FUNCTION_BLOCK Fb_SafetyCheck
VAR_INPUT
END_VAR
VAR_OUTPUT
END_VAR
VAR
	i, j:INT;
	m_checkDelay :ARRAY[1..g_maxNum] OF checkDelay;
	m_checkDelayTime :checkDelayTime;
	m_checkPermit:ARRAY[1..g_maxNum] OF  checkPermit;
	
	m_jntErrFlag:ARRAY[1..g_maxNum,0..g_maxArmJoint,1..3] OF BOOL;
	m_armErrFlag:ARRAY [1..g_maxNum,1..3] OF BOOL;
	m_errCode:UDINT;
	m_resetFlag : BOOL:= FALSE;
	m_resetFlagTon : TON;
	
	m_errNumType: ARRAY [1..3] OF INT;
	m_ArrayErrCodeType:ARRAY [1..3] OF ARRAY [0..100] OF UDINT;
	
	//The fault is sent to the UI at the frequency of 0.1S
	m_errCodeUpdateFlag: ARRAY [1..3] OF BOOL;
	m_errCodeUpdateTon: ARRAY [1..3] OF TON;
	
	m_curJntTorqueIOlast :ARRAY [1..g_maxArmNum] OF vec7di;  
	m_cmdJntPosLast : ARRAY [1..g_maxArmNum] OF vec7d;  
	m_cartCurJntTorqueIOlast :ARRAY [1..4] OF LREAL;  
	m_cartCmdJntPosLast : ARRAY [1..4] OF LREAL; 
	o_ErrCode:ARRAY [1..3] OF UDINT;
		
	//error robot data record
	m_dataRecord : Fb_dataRecord;
	
	m_PromptMassBusy:BOOL;
	m_PromptFlag:ARRAY[1..g_maxNum,1..20] OF UINT;
	m_deleteCode:UDINT;
	m_EtherCATCheck :ARRAY [1..g_mArmNum] OF Fb_EtherCATCheck;
	
	//drive  heartbeat single check
	m_heartbeatCheck :ARRAY [1..g_maxNum] OF ARRAY [1..g_maxArmJoint] OF FB_HeartbeatDetect;
	m_bHeartbeatCheck : ARRAY [1..g_maxNum] OF ARRAY [1..g_maxArmJoint] OF BOOL;
END_VAR


VAR CONSTANT
	m_codeUpdateDelay:TIME:=T#0.1S;
	
	//Fault level: 1 indicates  prompt message, 2 indicates a recoverable fault and 3 indicates an unrecoverable fault
	m_promptMessageLevel : UINT :=1;
	m_rcvLevel : UINT :=2;
	m_unrcvLevel : UINT :=3;
END_VAR


METHOD armSafetyCheck : BOOL
VAR_INPUT
	i_armId:INT;
	i_safetyCheckVar :ARRAY[1..g_maxNum] OF checkInputVariable;
	i_masterStatus :ST_MasterStatus;
	i_masterJointData : ST_MasterJointData;
END_VAR

VAR
	k:INT;
	motorHallCheck : UDINT;
	motorPhaseCheck : UDINT;
	motorDriveError : BOOL;
	lossCommuniJoint : INT;
END_VAR
//驱动器状态监测、驱动器未连接
FOR i:=1 TO g_mJntNum BY 1 DO
	m_bHeartbeatCheck[i_armId][i] := TRUE;//m_heartbeatCheck[i_armId][i].run(i_safetyCheckVar[i_armId].m_masterDriverInput[i].m_heartBeat);
	m_checkDelay[i_armId].T_jntStatusErr[i](IN:= (i_safetyCheckVar[i_armId].m_masterDriverInput[i].m_statusWord=0 AND m_checkPermit[i_armId].m_jntStatusErr[i]), PT:=m_checkDelayTime.Ti_jntStatusErr , Q=> , ET=> );
	IF m_checkDelay[i_armId].T_jntStatusErr[i].Q OR NOT m_bHeartbeatCheck[i_armId][i] THEN
		errCodeAssign(i_armId, i_armId,  0, i, 16#3002 ,m_unrcvLevel );
		EXIT;
	END_IF
END_FOR



//关节编码器监测
FOR i:=1 TO g_mJntNum BY 1 DO	
	IF i = 2 THEN
		//m_checkDelay[i_ArmId].T_linkEncErrCode[i](IN:= (driveErrorCheck(i_armId, i, 1, i_safetyCheckVar[i_ArmId].m_masterDriverInput[4].m_driverError) > 0  AND m_checkPermit[i_ArmId].m_linkEncErr[i]), PT:=m_checkDelayTime.Ti_linkEncErrCode , Q=> , ET=> );
	ELSE
		//m_checkDelay[i_ArmId].T_linkEncErrCode[i](IN:= (driveErrorCheck(i_armId, i, 1, i_safetyCheckVar[i_ArmId].m_masterDriverInput[i].m_driverError) > 0  AND m_checkPermit[i_ArmId].m_linkEncErr[i]), PT:=m_checkDelayTime.Ti_linkEncErrCode , Q=> , ET=> );
	END_IF
	m_checkDelay[i_ArmId].T_linkEncErr[i](IN:= (i_safetyCheckVar[i_ArmId].m_masterDriverInput[i].m_linkEncoder=g_maxLinkEnc OR i_safetyCheckVar[i_ArmId].m_masterDriverInput[i].m_linkEncoder=g_minLinkEnc) AND m_checkPermit[i_ArmId].m_linkEncErr[i], PT:=m_checkDelayTime.Ti_linkEncErr , Q=> , ET=> );
	IF m_checkDelay[i_ArmId].T_linkEncErr[i].Q OR m_checkDelay[i_ArmId].T_linkEncErrCode[i].Q THEN
		errCodeAssign(i_ArmId, i_ArmId,  0, i,  16#3003 ,m_unrcvLevel );
	END_IF
END_FOR


//驱动器错误检测
//FOR i:=1 TO g_mJntNum BY 1 DO
//	m_checkDelay[i_ArmId].T_DriveErr[i](IN:= (i_safetyCheckVar[i_ArmId].m_masterDriverInput[i].m_driverError AND g_driveErrWord)=g_driveErrWord AND m_checkPermit[i_ArmId].m_driveErr[i] , PT:=m_checkDelayTime.Ti_driveErr , Q=> , ET=> );
//	IF m_checkDelay[i_ArmId].T_DriveErr[i].Q THEN
//		errCodeAssign(i_ArmId, i_ArmId,  0, i, 16#3004 ,m_unrcvLevel );
//	END_IF
//END_FOR


//双编码器偏差过大检测
FOR i:=1 TO g_mJntNum BY 1 DO
	m_checkDelay[i_ArmId].T_armJntEncErr[i](IN:= ABS(i_masterJointData.m_curLinkPos[i_armId][i]-i_masterJointData.m_curJntPos[i_armId][i])>=g_armMaxJntEncErr[i] AND m_checkPermit[i_ArmId].m_armJntEncErr[i], PT:=m_checkDelayTime.Ti_armJntEncErr , Q=> , ET=> );
	IF m_checkDelay[i_ArmId].T_armJntEncErr[i].Q THEN
		errCodeAssign( i_ArmId, i_ArmId,  0, i, 16#3005, m_unrcvLevel );
	END_IF
END_FOR


//关节运动超限位
FOR i:=1 TO g_mJntNum BY 1 DO
	m_checkDelay[i_armId].T_outOfLimit[i](IN:= (i_masterJointData.m_curJntPos[i_armId][i]>= (g_maxJntPos[i_armId,i] + g_armJntPosLimitBuffer[i]) OR i_masterJointData.m_curJntPos[i_armId][i]<=(g_minJntPos[i_armId,i] - g_armJntPosLimitBuffer[i])) AND m_checkPermit[i_ArmId].m_outOfLimit[i], PT:=m_checkDelayTime.Ti_outofLimit , Q=> , ET=> );
	IF m_checkDelay[i_armId].T_outOfLimit[i].Q THEN
		errCodeAssign(i_armId, i_ArmId,  0, i, 16#3006, m_unrcvLevel );
	END_IF
END_FOR

//check motor hall single, error code 27
FOR i:=1 TO g_mJntNum DO
	motorHallCheck := driveErrorCheck(i_armId, i, 2, i_safetyCheckVar[i_ArmId].m_masterDriverInput[i].m_driverError);		
	m_checkDelay[i_ArmId].T_motorHallCheck[i](IN:= (motorHallCheck  = 1) , PT:=m_checkDelayTime.Ti_motorHallCheck , Q=> , ET=> );
	IF  m_checkDelay[i_ArmId].T_motorHallCheck[i].Q THEN
		errCodeAssign(i_ArmId, i_ArmId,  0, i, 16#300B ,m_unrcvLevel );
	END_IF
END_FOR


//check motor phase single, error code 30
FOR i:=1 TO g_mJntNum DO
	motorPhaseCheck := driveErrorCheck(i_armId, i, 3, i_safetyCheckVar[i_ArmId].m_masterDriverInput[i].m_driverError);		
	m_checkDelay[i_ArmId].T_motorPhaseCheck[i](IN:= (motorPhaseCheck  = 1) , PT:=m_checkDelayTime.Ti_motorPhaseCheck , Q=> , ET=> );
	IF  m_checkDelay[i_ArmId].T_motorPhaseCheck[i].Q THEN
		errCodeAssign(i_ArmId, i_ArmId,  0, i, 16#300C ,m_unrcvLevel );
	END_IF
END_FOR


//check motor drive, error code 31
FOR i:=1 TO g_mJntNum DO
	motorDriveError := (i_safetyCheckVar[i_ArmId].m_masterDriverInput[i].m_driverError AND 16#80000000)=16#80000000;
	m_checkDelay[i_ArmId].T_motorDriveError[i](IN:= motorDriveError, PT:=m_checkDelayTime.Ti_motorDriveCheck , Q=> , ET=> );
	IF  m_checkDelay[i_ArmId].T_motorDriveError[i].Q THEN
		errCodeAssign(i_ArmId, i_ArmId,  0, i, 16#300D ,m_unrcvLevel );
	END_IF
END_FOR


//关节跟随误差过大
FOR i:=1 TO g_mJntNum BY 1 DO
	m_checkDelay[i_ArmId].T_armJntFollowErr[i](IN:= ABS(i_masterJointData.m_cmdJntPos[i_armId][i]- i_masterJointData.m_curJntPos[i_armId][i])>g_armMaxJntFollowErr[i]  AND m_checkPermit[i_ArmId].m_armJntFollowErr[i], PT:=m_checkDelayTime.Ti_armJntFollowErr , Q=> , ET=> );
	IF m_checkDelay[i_ArmId].T_armJntFollowErr[i].Q THEN
		errCodeAssign(i_ArmId, i_ArmId,  0, i, 16#2002, m_rcvLevel );
	END_IF
END_FOR


//笛卡尔空间指令与位置偏差检测
//FOR i:=1 TO 6 BY 1 DO
//	m_checkDelay[i_ArmId].T_spacePoseErr[i](IN:= i_safetyCheckVar[i_ArmId].m_spacePoseErr[i]> g_maxCartPoseErr[i] AND m_checkPermit[i_ArmId].m_spacePoseErr[i], PT:=m_checkDelayTime.Ti_spacePoseErr , Q=> , ET=> );
//	IF m_checkDelay[i_ArmId].T_spacePoseErr[i].Q THEN
//		errCodeAssign(i_ArmId, i_ArmId, 1, i, 16#2004, m_rcvLevel );
//	END_IF
//END_FOR


//current overrun check
FOR i:=1 TO g_mJntNum BY 1 DO
	m_checkDelay[i_armId].T_jntCurrentErr[i](IN:= ABS(i_safetyCheckVar[i_armId].m_motorCurrentIntegral[i])>g_motorCurrentLimit[i] AND m_checkPermit[i_ArmId].m_jntCurrentErr[i], PT:=m_checkDelayTime.Ti_jntCurrentErr , Q=> , ET=> );
	IF m_checkDelay[i_armId].T_jntCurrentErr[i].Q THEN
		errCodeAssign(i_armId, i_ArmId,  0, i, 16#2005, m_rcvLevel );
	END_IF
END_FOR


//Ethercat communication check
lossCommuniJoint := g_maxArmJoint;
FOR i:=1 TO g_mJntNum BY 1 DO
	IF NOT i_safetyCheckVar[i_ArmId].m_EtherCATState[i].EtherCATState THEN
		lossCommuniJoint := MIN(lossCommuniJoint,i);
		errCodeAssign(i_ArmId, i_ArmId, 0, lossCommuniJoint, 16#2006, m_rcvLevel );
		IF i > lossCommuniJoint THEN
			m_jntErrFlag[i_armId,i,m_rcvLevel]:=TRUE;
		END_IF
	END_IF
END_FOR


//self check failure
IF i_masterStatus.m_armState[i_armId] = MasterArmState_Home AND i_masterStatus.m_timePeriod[i] > g_selfCheckTimeLimit THEN//i_safetyCheckVar[i_armId].m_selfCheckFail THEN
	errCodeAssign(i_armId, i_ArmId,  0, 0, 16#2010, m_rcvLevel );
END_IF

//motor encoder mutation detection
FOR i:=1 TO g_mJntNum BY 1 DO
	IF i_safetyCheckVar[i_armId].m_motorEncSaltaValue[i]>g_maxJntCurSalta[i] THEN
		errCodeAssign(i_armId, i_ArmId, 0, i, 16#200C, m_rcvLevel );
	END_IF
END_FOR

//master hall anomaly
IF i_masterStatus.m_gripHallSensor[i_armId] = 0 THEN
	errCodeAssign(i_armId, i_ArmId, 0, 0, 16#200E, m_rcvLevel );
END_IF

//drive Ethercat CRC lost
FOR i:=1 TO g_mJntNum BY 1 DO
	IF (i_safetyCheckVar[i_armId].m_EtherCATState[i].CRCPortA)>m_minLossFrame OR  (i_safetyCheckVar[i_armId].m_EtherCATState[i].CRCPortB)>m_minLossFrame OR  (i_safetyCheckVar[i_armId].m_EtherCATState[i].CRCPortC)>m_minLossFrame  THEN
		errCodeAssign(i_armId, i_ArmId, 0, i, 16#200F, m_rcvLevel );
	END_IF
END_FOR
END_METHOD

METHOD arrayDeleteFrist : ARRAY [0..100] OF UDINT;
VAR_INPUT
	i_array:ARRAY [0..100] OF UDINT;
END_VAR

VAR
	k:INT;
END_VAR

arrayDeleteFrist[100]:=0;

FOR k:=0 TO 99 BY 1 DO
	arrayDeleteFrist[k]:=i_array[k+1];
END_FOR
END_METHOD

METHOD arrayDeleteInput : BOOL
VAR_INPUT
	i_Array:ARRAY[0..100] OF UDINT;
	i_DeleteCode:UDINT;
END_VAR

VAR_OUTPUT
	o_Array:ARRAY[0..100] OF UDINT;
	
END_VAR

VAR
	i:INT;
	Falg:BOOL;
END_VAR

FOR i:=0 TO 20 BY 1 DO 
	IF i_Array[i]=i_DeleteCode THEN
		Falg:=TRUE;
	END_IF
	
	IF Falg=TRUE THEN
		o_Array[i]:=i_Array[i+1];
	ELSE
		o_Array[i]:=i_Array[i];
	END_IF
END_FOR
o_Array[20]:=0;
END_METHOD

METHOD arrayFIFO : ARRAY [0..100] OF  UDINT
VAR_INPUT
	i_array:ARRAY[0..100] OF UDINT;
	i_newData:UDINT;
END_VAR

VAR
	i:INT;
END_VAR

FOR i:=0 TO 20 BY 1 DO
	arrayFIFO[i+1]:=i_array[i];
END_FOR

arrayFIFO[0]:=i_newData;
END_METHOD

METHOD arrayFILO : ARRAY [0..100] OF  UDINT
VAR_INPUT
	i_array:ARRAY[0..100] OF UDINT;
	i_newData:UDINT;
END_VAR

VAR
	i:INT;
END_VAR

FOR i:=0 TO 99 BY 1 DO
	arrayFILO[i]:=i_array[i];
	IF i_array[i]=0 THEN
		arrayFILO[i]:=i_newData;
		EXIT;
	END_IF
END_FOR
END_METHOD

METHOD cartSafetyCheck : BOOL
VAR_INPUT
	i_armId:INT;
	i_safetyCheckVar : checkInputVariable;
	i_cartJointData : ST_CartJointData;
END_VAR


VAR
	k:INT;
	motorHallCheck : UDINT;
	motorPhaseCheck : UDINT;
	motorDriveError : BOOL;
	lossCommuniJoint : INT;
END_VAR
//驱动器状态监测、驱动器未连接
FOR i:=1 TO g_maxCartJoint BY 1 DO
	m_bHeartbeatCheck[i_armId][i] := TRUE;//m_heartbeatCheck[i_armId][i].run(i_safetyCheckVar.m_cartDriverInput[i].m_heartBeat);
	m_checkDelay[i_armId].T_cartJntStatusErr[i](IN:= (i_safetyCheckVar.m_cartDriverInput[i].m_statusWord=0 AND m_checkPermit[i_ArmId].m_cartJntStatus[i]), PT:=m_checkDelayTime.Ti_CarJntStatus , Q=> , ET=> );
	IF m_checkDelay[i_armId].T_cartJntStatusErr[i].Q OR NOT m_bHeartbeatCheck[i_armId][i] THEN
		errCodeAssign(i_armId, i_ArmId,  0, i, 16#3002 ,m_unrcvLevel );
	END_IF
END_FOR



//关节编码器监测
FOR i:=1 TO g_maxCartJoint BY 1 DO
	m_checkDelay[i_ArmId].T_cartLinkEncErrCode[i](IN:= (driveErrorCheck(i_armId, i, 1, i_safetyCheckVar.m_cartDriverInput[i].m_driverError) > 0  AND m_checkPermit[i_ArmId].m_linkEncErr[i]), PT:=m_checkDelayTime.Ti_linkEncErrCode , Q=> , ET=> );
	m_checkDelay[i_armId].T_cartLinkEncErr[i](IN:= (i_safetyCheckVar.m_cartDriverInput[i].m_linkEncoder=g_cartMaxLinkEnc[i] OR i_safetyCheckVar.m_cartDriverInput[i].m_linkEncoder=g_cartMinLinkEnc[i]) AND m_checkPermit[i_ArmId].m_cartJntEncErr[i], PT:=m_checkDelayTime.Ti_CarActSec , Q=> , ET=> );
	IF m_checkDelay[i_ArmId].T_cartLinkEncErrCode[i].Q OR m_checkDelay[i_armId].T_cartLinkEncErr[i].Q THEN
		errCodeAssign(i_armId, i_ArmId,  0, i, 16#3003 ,m_unrcvLevel );
	END_IF
END_FOR


////驱动器错误检测
//FOR i:=1 TO g_maxCartJoint BY 1 DO
//	m_checkDelay[i_armId].T_cartDriveErr[i](IN:= (i_safetyCheckVar.m_cartDriverInput[i].m_driverError AND g_driveErrWord)=g_driveErrWord AND m_checkPermit[i_ArmId].m_cartDriveErr[i] , PT:=m_checkDelayTime.Ti_CarDriveErr , Q=> , ET=> );
//	IF m_checkDelay[i_armId].T_cartDriveErr[i].Q THEN
//		errCodeAssign(i_armId, i_ArmId,  0, i, 16#3004 ,m_unrcvLevel );
//	END_IF
//END_FOR



//台车双编码器偏差过大
FOR i:=1 TO g_maxCartJoint BY 1 DO
	m_checkDelay[i_armId].T_cartJntEncErr[i](IN:= ABS (i_cartJointData.m_curLinkPos[i]-i_cartJointData.m_curJntPos[i])>g_cartMaxJntEncErr[i] AND m_checkPermit[i_ArmId].m_cartJntEncErr[i], PT:=m_checkDelayTime.Ti_CarDualEncDev , Q=> , ET=> );
	IF m_checkDelay[i_armId].T_cartJntEncErr[i].Q THEN
		errCodeAssign(i_armId, i_ArmId,  0, i, 16#3005 ,m_unrcvLevel );
	END_IF
END_FOR


//关节运动超限位
FOR i:=1 TO g_maxCartJoint BY 1 DO
	m_checkDelay[i_armId].T_cartOutOfLimit[i](IN:= (i_cartJointData.m_curJntPos[i]>=g_cartMaxJntLimit[i] OR i_cartJointData.m_curJntPos[i]<=g_cartMinJntLimit[i]) AND m_checkPermit[i_ArmId].m_cartOutOfLimit[i] , PT:=m_checkDelayTime.Ti_CaroutofLimit , Q=> , ET=> );
	IF m_checkDelay[i_armId].T_cartOutOfLimit[i].Q THEN
		errCodeAssign(i_armId, i_ArmId,  0, i, 16#3006 ,m_unrcvLevel );
	END_IF
END_FOR

//check motor hall single, error code 27
FOR i:=1 TO g_maxCartJoint DO
	motorHallCheck := driveErrorCheck(i_armId, i, 2, i_safetyCheckVar.m_cartDriverInput[i].m_driverError);		
	m_checkDelay[i_ArmId].T_cartMotorHallCheck[i](IN:= (motorHallCheck  = 1) , PT:=m_checkDelayTime.Ti_carMotorHallCheck , Q=> , ET=> );
	IF  m_checkDelay[i_ArmId].T_cartMotorHallCheck[i].Q THEN
		errCodeAssign(i_ArmId, i_ArmId,  0, i, 16#300B ,m_unrcvLevel );
	END_IF
END_FOR


//check motor phase single, error code 30
FOR i:=1 TO g_maxCartJoint DO
	motorPhaseCheck := driveErrorCheck(i_armId, i, 3,i_safetyCheckVar.m_cartDriverInput[i].m_driverError);			
	m_checkDelay[i_ArmId].T_cartMotorPhaseCheck[i](IN:= (motorPhaseCheck  = 1) , PT:=m_checkDelayTime.Ti_carMotorPhaseCheck , Q=> , ET=> );
	IF  m_checkDelay[i_ArmId].T_cartMotorPhaseCheck[i].Q THEN
		errCodeAssign(i_ArmId, i_ArmId,  0, i, 16#300C ,m_unrcvLevel );
	END_IF
END_FOR


//check motor drive, error code 31
FOR i:=1 TO g_maxCartJoint DO
	motorDriveError := (i_safetyCheckVar.m_cartDriverInput[i].m_driverError AND 16#80000000)=16#80000000;
	m_checkDelay[i_ArmId].T_cartMotorDriveError[i](IN:= motorDriveError, PT:=m_checkDelayTime.Ti_carMotorDriveCheck , Q=> , ET=> );
	IF  m_checkDelay[i_ArmId].T_cartMotorDriveError[i].Q THEN
		errCodeAssign(i_ArmId, i_ArmId,  0, i, 16#300D ,m_unrcvLevel );
	END_IF
END_FOR

//关节跟随误差过大
FOR i:=1 TO g_maxCartJoint BY 1 DO
	m_checkDelay[i_armId].T_cartJntFollowErr[i](IN:= ABS(i_cartJointData.m_cmdJntPos[i]- i_cartJointData.m_curJntPos[i])>g_cartMaxJntFollowErr[i]  AND m_checkPermit[i_ArmId].m_cartFollowErr[i], PT:=m_checkDelayTime.Ti_CarFollowDev , Q=> , ET=> );
	IF m_checkDelay[i_armId].T_cartJntFollowErr[i].Q THEN
		errCodeAssign(i_armId, i_ArmId,  0, i, 16#2002 ,m_rcvLevel );
	END_IF
END_FOR


//关节速度监控
FOR i:=1 TO g_maxCartJoint BY 1 DO
	m_checkDelay[i_armId].T_cartJntVelErr[i](IN:= ABS(i_cartJointData.m_curJntVel[i])>g_cartMaxJntVel[i] AND m_checkPermit[i_ArmId].m_cartJntVelErr[i], PT:=m_checkDelayTime.Ti_CarJntVel , Q=> , ET=> );
	IF m_checkDelay[i_armId].T_cartJntVelErr[i].Q THEN
		errCodeAssign(i_armId, i_ArmId,  0, i, 16#2003 ,m_rcvLevel );
	END_IF
END_FOR


//电流超限监测
FOR i:=1 TO g_maxCartJoint BY 1 DO
	m_checkDelay[i_armId].T_cartJntCurrentErr[i](IN:= ABS(i_cartJointData.m_curJntTrq[i])>g_cartMaxJntCurrent[i] AND m_checkPermit[i_ArmId].m_cartJntCurrentErr[i], PT:=m_checkDelayTime.Ti_CarJntCurrent , Q=> , ET=> );
	IF m_checkDelay[i_armId].T_cartJntCurrentErr[i].Q THEN
		errCodeAssign(i_armId, i_ArmId,  0, i, 16#2005 ,m_rcvLevel );
	END_IF
END_FOR


//Ethercat通讯检测
lossCommuniJoint := g_maxCartJoint;
FOR i:=1 TO g_maxCartJoint BY 1 DO
	IF NOT i_safetyCheckVar.m_cartEtherCATState[i].EtherCATState THEN
		lossCommuniJoint := MIN(lossCommuniJoint,i);
		errCodeAssign(i_ArmId, i_ArmId,  0, lossCommuniJoint, 16#2006 ,m_rcvLevel );
		IF i > lossCommuniJoint THEN
			m_jntErrFlag[i_armId,i,m_rcvLevel]:=TRUE;
		END_IF
	END_IF
END_FOR
END_METHOD

METHOD checkOPStatus : UDINT
VAR_IN_OUT CONSTANT
	i_armEtherCATOPStatus :vec2b;
	i_cartEtherCATOPStatus : BOOL;
END_VAR
VAR
	arm : UDINT;
END_VAR

VAR_STAT
	clearFaultTime : FB_TON;
END_VAR
FOR arm := 1 TO g_mArmNum DO
	IF NOT i_armEtherCATOPStatus[arm] THEN
		checkOPStatus:=SHL(arm,24)+SHL(0,16)+16#2010;
		g_ArrayErrCodeArm[arm][0] := checkOPStatus;
		EXIT;
	END_IF
END_FOR

IF NOT i_cartEtherCATOPStatus THEN
	checkOPStatus:=SHL(g_cartNum,24)+SHL(0,16)+16#2011;
	g_ArrayErrCodeArm[g_cartNum][0] := checkOPStatus;
END_IF

clearFaultTime(IN:=  GVL_interactUI.g_uiResetFault=1, PT:= T#150MS, Q=> , ET=> );
IF GVL_interactUI.g_uiResetFault=1 THEN
	checkOPStatus := 0;
	IF clearFaultTime.Q THEN
		GVL_interactUI.g_uiResetFault:=0;
	END_IF
END_IF
END_METHOD

PROPERTY checkPermit : REFERENCE TO ARRAY[1..g_maxNum] OF  checkPermit
GET
checkPermit ref= m_checkPermit;
END_GET
SET
END_SET
END_PROPERTY

METHOD driveErrorCheck : UDINT
VAR_INPUT
	i_armId:INT;
	i_jntId :INT;
	i_checkMode : INT;//1 link encoder error ,2 motor hall error, 3 motor phase loss 
	i_driverError :UDINT;
END_VAR
VAR
	driveErrMassage : UDINT;
	errorTemp :ARRAY [1..3] OF UDINT; //check mode number
	checkMode : INT;
	encErrorJnt : ARRAY [1..3] OF UDINT;
	motorHallErrorJnt : ARRAY [1..3] OF UDINT;
	motorPhaseLossJnt : ARRAY [1..3] OF UDINT;
END_VAR
driveErrMassage := i_driverError;
encErrorJnt[1] := SHR(driveErrMassage,6) AND 16#07;
encErrorJnt[2] := SHR(driveErrMassage,9) AND 16#07;
encErrorJnt[3] := SHR(driveErrMassage,12) AND 16#07;
motorHallErrorJnt[2] := SHR(driveErrMassage,22) AND 16#01;
motorPhaseLossJnt[2] := SHR(driveErrMassage,23) AND 16#01;
motorHallErrorJnt[1] := SHR(driveErrMassage,27) AND 16#01;
motorPhaseLossJnt[1] := SHR(driveErrMassage,30) AND 16#01;

IF i_armId <= g_sArmNum THEN
	IF i_jntId = 2  THEN
		errorTemp[1] :=encErrorJnt[2];
		errorTemp[2] :=motorHallErrorJnt[2];
		errorTemp[3] :=motorPhaseLossJnt[2];
	ELSE
		errorTemp[1] :=encErrorJnt[1];
		errorTemp[2] :=motorHallErrorJnt[1];
		errorTemp[3] :=motorPhaseLossJnt[1];
	END_IF
ELSE
	errorTemp[1] :=encErrorJnt[1];
	errorTemp[2] :=motorHallErrorJnt[1];
	errorTemp[3] :=motorPhaseLossJnt[1];
END_IF
checkMode := LIMIT (1, i_checkMode, 3);
driveErrorCheck := errorTemp[checkMode];
END_METHOD

METHOD electriAngleDev : DINT
VAR_INPUT
	i_motorElectriAngleDev : DINT;
END_VAR

IF i_motorElectriAngleDev > 50000 THEN
	electriAngleDev := i_motorElectriAngleDev - 65535;
ELSIF i_motorElectriAngleDev < -50000 THEN
	electriAngleDev := i_motorElectriAngleDev + 65535;
ELSE
	electriAngleDev := i_motorElectriAngleDev;
END_IF
END_METHOD

METHOD errCodeAssign : BOOL
VAR_INPUT
	i_armId:UDINT;
	i_errLocation:UDINT;
	i_errCodeMode:UDINT;
	i_errJoint:UDINT;
	i_errID:UDINT;
	i_errFlagID :UINT;
END_VAR
IF m_jntErrFlag[i_armId,i_errJoint,i_errFlagID]=FALSE THEN
	m_jntErrFlag[i_armId,i_errJoint,i_errFlagID]:=TRUE;
	m_errCode:=SHL(i_errLocation,24)+SHL(i_errCodeMode,20)+SHL(i_errJoint,16)+i_errID;
	
	
	IF i_errID>=16#3000 THEN
		m_errNumType[m_unrcvLevel]:=LIMIT(0,m_errNumType[m_unrcvLevel]+1,100);
		m_arrayErrCodeType[m_unrcvLevel][m_errNumType[m_unrcvLevel]]:=m_errCode;
		g_arrayErrCodeArm[i_armId]:=arrayFILO(i_Array:= g_arrayErrCodeArm[i_ArmId], i_NewData:=m_errCode );
		m_armErrFlag[i_armId,m_unrcvLevel]:=TRUE;
		
	ELSIF i_errID>=16#2000 THEN
		m_errNumType[m_rcvLevel]:=LIMIT(0,m_errNumType[m_rcvLevel]+1,100);
		m_arrayErrCodeType[m_rcvLevel][m_errNumType[m_rcvLevel]]:=m_errCode;
		g_arrayErrCodeArm[i_armId]:=arrayFILO(i_Array:= g_arrayErrCodeArm[i_ArmId], i_NewData:=m_errCode );
		m_armErrFlag[i_armId,m_rcvLevel]:=TRUE;
		
	END_IF
END_IF
END_METHOD

METHOD errCodeUpdating :ARRAY [1..3] OF UDINT;
VAR_INPUT
END_VAR

m_errCodeUpdateTon[m_unrcvLevel](IN:= NOT m_errCodeUpdateFlag[3], PT:=m_codeUpdateDelay , Q=> m_errCodeUpdateFlag[3], ET=> );
IF m_errCodeUpdateFlag[m_unrcvLevel] THEN
	IF m_errNumType[m_unrcvLevel]>=1 THEN
		m_ArrayErrCodeType[m_unrcvLevel]:=ArrayDeleteFrist(i_Array:=m_ArrayErrCodeType[3]) ;
		o_ErrCode[m_unrcvLevel]:=m_ArrayErrCodeType[m_unrcvLevel][0] ;
		g_ArrayErrCodeTypeTest[m_unrcvLevel]:=arrayFILO(i_Array:= g_ArrayErrCodeTypeTest[m_unrcvLevel], i_NewData:=o_ErrCode[m_unrcvLevel] );
		m_errNumType[m_unrcvLevel]:=m_errNumType[m_unrcvLevel]-1;
	END_IF
END_IF


m_errCodeUpdateTon[m_rcvLevel](IN:= NOT m_errCodeUpdateFlag[2], PT:=m_codeUpdateDelay , Q=> m_errCodeUpdateFlag[2], ET=> );
IF m_errCodeUpdateFlag[m_rcvLevel] THEN
	IF m_errNumType[m_rcvLevel]>=1 THEN
		m_ArrayErrCodeType[m_rcvLevel]:=ArrayDeleteFrist(i_Array:=m_ArrayErrCodeType[m_rcvLevel]) ;
		o_ErrCode[m_rcvLevel]:=m_ArrayErrCodeType[m_rcvLevel][0] ;
		g_ArrayErrCodeTypeTest[m_rcvLevel]:=arrayFILO(i_Array:= g_ArrayErrCodeTypeTest[m_rcvLevel], i_NewData:=o_ErrCode[m_rcvLevel] );
		m_errNumType[m_rcvLevel]:=m_errNumType[m_rcvLevel]-1;
	END_IF
END_IF
END_METHOD

METHOD errFlagReset : BOOL
VAR_INPUT
END_VAR
FOR i := 1 TO g_maxNum DO
	FOR j :=0 TO g_maxArmJoint DO
		m_jntErrFlag[i, j, 2]:=FALSE;
	END_FOR
	m_armErrFlag[i, 2]:=FALSE;
END_FOR

FOR i := 1 TO g_mArmNum DO
	m_EtherCATCheck[i].clearCRCError(GVL_SystemParameters.g_masterArmNetID[i]);
END_FOR

m_ArrayErrCodeType[2] := g_zeroErrCodeArray;
m_resetFlag := TRUE;
o_ErrCode[2]:=0;
END_METHOD

METHOD poseErrCheck : vec6d
VAR_INPUT
	i_cmdPose : ST_Frame;
	i_curPose :ST_Frame;
END_VAR

VAR
	posErr,oriErr:Vec3d;
	matT,rotErr:Mat3d;
	errAngle :LREAL;
	errAxis :Vec3d;
	i : INT;
END_VAR
vecSub(i_cmdPose.m_pos, i_curPose.m_pos,posErr);

matTranspose(i_cmdPose.m_rot, matT);
matMultiply(matT,i_curPose.m_rot, rotErr);
rot2AngAxis(rotErr, angle=>errAngle, axis=>errAxis);
vecMultiNum(errAxis, errAngle,oriErr);

FOR i := 1 TO 6 DO
	IF i <= 3 THEN
		poseErrCheck[i] := posErr[i];
	ELSE
		poseErrCheck[i] := oriErr[i];
	END_IF
END_FOR
END_METHOD

METHOD promptMassCode : BOOL
VAR_INPUT
	i_PromptStatus:BOOL;
	i_ArmId:UDINT;
	i_ErrID:UDINT;
	i_ErrLocation:UDINT;
END_VAR

m_PromptMassBusy:=TRUE;

//提示置位
IF i_PromptStatus=TRUE AND m_PromptFlag[i_ArmId,i_ErrID]=0 THEN
	m_PromptFlag[i_ArmId,i_ErrID]:=1;
END_IF

//输出提示故障码
IF m_PromptFlag[i_ArmId,i_ErrID]=1 THEN
	m_ErrCode:=SHL(i_ErrLocation,24)+i_ErrID+16#1010;
	m_ArrayErrCodeType[1]:=ArrayFIFO(i_Array:= m_ArrayErrCodeType[1], i_NewData:=m_ErrCode );//m_ErrCode;
	m_PromptFlag[i_ArmId,i_ErrID]:=2;
END_IF

//清除提示故障码
IF m_PromptFlag[i_ArmId,i_ErrID]=2 AND i_PromptStatus=FALSE THEN
	m_deleteCode:=SHL(i_ErrLocation,24)+i_ErrID+16#1010;
	ArrayDeleteInput(i_Array:= m_ArrayErrCodeType[1], i_DeleteCode:=m_deleteCode , o_Array=> m_ArrayErrCodeType[1]);
	m_PromptFlag[i_ArmId,i_ErrID]:=0;
END_IF
o_ErrCode[1]:=m_ArrayErrCodeType[1][0];
m_PromptMassBusy:=FALSE;
END_METHOD

METHOD systemSafetyCheck : BOOL
VAR_INPUT
	i_armId:INT;
	i_safetyCheckVar :ARRAY[1..g_maxNum] OF checkInputVariable;
	i_masterStatus :ST_MasterStatus;
	i_cartJointData : ST_CartJointData;
	i_masterJointData : ST_MasterJointData;
END_VAR

VAR
	k:INT;
END_VAR
m_resetFlagTon(IN:= m_resetFlag, PT:= T#0.1S, Q=> , ET=> );
IF m_resetFlagTon.Q THEN
	m_resetFlag := FALSE;
END_IF
IF m_resetFlag THEN
	RETURN;
END_IF


IF i_armId =g_cartNum THEN 
	//cart safrty check
	cartSafetyCheck(i_armId,i_safetyCheckVar[i_armId],i_cartJointData);
ELSE
	//master arms safety check
	armSafetyCheck(i_armId,i_safetyCheckVar,i_masterStatus,i_masterJointData);
END_IF

//StopButton
IF  i_safetyCheckVar[i_ArmId].PCStopButton=0 OR NOT i_safetyCheckVar[i_ArmId].MasterStopButton OR i_safetyCheckVar[i_ArmId].SlaveStopButton THEN
	errCodeAssign(i_ArmId, 16#0B, 0, 0, 16#2001, m_rcvLevel );
END_IF

//prompt message
FOR i:=1 TO 10 DO
	PromptMassCode( i_safetyCheckVar[i_ArmId].m_promptStatus[i], i_ArmId,  i,  i_safetyCheckVar[i_ArmId].m_promptLocation[i]);
END_FOR
END_METHOD

END_FUNCTION_BLOCK

(* stored: Version 1.1.0.1, ProductVersion 3.1.4024.11
   POU Fb_SafetyCheck: Id {d7e5b419-2971-4dae-96a7-39fe3a1a6245}, SpecialFunc None
   Folder interface: Id {17cc820b-439e-4bcd-b035-470b65e01b6b}
   Method armSafetyCheck: Id {1102e175-6107-4706-a6ad-ea5e8fc76a1b}
   Method arrayDeleteFrist: Id {00e49c9f-cbe8-4b26-b05a-c4b6acb31969}
   Method arrayDeleteInput: Id {980f1673-9d6d-4af2-a068-78f386b10642}
   Method arrayFIFO: Id {655e2224-db9d-4b4a-8461-cda6c8a0a0dc}
   Method arrayFILO: Id {26262d95-ef1c-497d-b548-c28fcd1771c9}
   Method cartSafetyCheck: Id {64489d60-54d3-406d-a82e-df5d6a98f0f1}
   Method checkOPStatus: Id {3d1e8b99-1cb7-4b50-92fc-5aa7708cc80d}
   Property checkPermit: Id {4ac5d9ef-e4e1-4258-a3b3-a263171adb15}
   Get Get: Id {5a600670-0a2f-4560-9a82-9a30fff97e6d}
   Set Set: Id {06536298-2ca0-4bed-b4ee-b29089d28252}
   Method driveErrorCheck: Id {4528636a-c0d4-42b4-803c-17712e93425f}
   Method electriAngleDev: Id {8c2ea40a-ba18-4d9e-8d1f-4ea5c9f320b3}
   Method errCodeAssign: Id {c6bfedc5-fddc-4db6-ba7d-64971d20a433}
   Method errCodeUpdating: Id {0b3c9bb2-9217-4fc9-b998-e4a685172889}
   Method errFlagReset: Id {2f8c115b-de2b-4c35-92d2-fdbed32dcf1f}
   Method poseErrCheck: Id {634b1f68-028c-4865-89df-6d37274cf53c}
   Method promptMassCode: Id {97898266-aa01-4d86-bccd-f23152d91670}
   Method systemSafetyCheck: Id {7874ef26-88d5-4eb7-8db9-4fa17a2dd1f0} *)
